Yaskawa INFORM job: R1_W70(-90,-90)KM-OK.JBI

/JOB
//NAME R1_W70(-90,-90)KM-OK
///FOLDERNAME KRIS-SCIANA
//POS
///NPOS 26,26,0,2,0,0
///TOOL 0
///POSTYPE PULSE
///PULSE
C00000=-196132,-11022,-16930,-25184,110789,12941
C00001=-198011,-10214,-12875,-25246,108327,12753
C00002=-198761,-9802,-11178,-25280,107342,12679
C00003=-197276,-7083,-6529,-24728,106458,13461
C00004=-197885,-7685,-6161,-24792,105787,13370
C00005=-197276,-7083,-6529,-24728,106458,13461
C00006=-198761,-9802,-11178,-25280,107342,12679
C00007=-193286,-14380,-9313,-33730,103593,14681
C00008=-192731,-13207,-7474,-33533,103368,14984
C00009=-193286,-14380,-9313,-33730,103593,14681
C00010=-191707,-12912,-9048,-33504,104715,14994
C00011=-204462,-13583,-17636,-16762,111010,11194
C00012=-206397,-14791,-14673,-16969,108266,10864
C00013=-206838,-12872,-13205,-17089,108253,10699
C00014=-206397,-14791,-14673,-16969,108266,10864
C00015=-200372,-41682,-38258,-22199,95841,14932
C00016=-196030,-47223,-44082,-25836,85574,-59294
C00017=-191753,-48190,-35047,-35552,77646,-65721
C00018=-174564,-4070,22503,-61552,98603,-65138
C00019=-192317,-48759,-35103,-35538,77200,-65811
C00020=-191548,-47635,-34025,-35606,77450,-65570
C00021=-178158,2617,28057,-62538,96414,-65728
C00022=-181749,10561,34999,-63443,94109,-66210
C00023=-190949,-52196,-43416,-35314,80525,-66319
C00024=-185515,-44796,-41028,-35596,84702,-65414
C00025=-121469,-118811,-94940,-10750,50157,59467
BC00000=386246,15,1075175
BC00001=386246,15,1075175
BC00002=386246,15,1075175
BC00003=386246,15,1075175
BC00004=386246,15,1075175
BC00005=386246,15,1075175
BC00006=386246,15,1075175
BC00007=386246,15,1075175
BC00008=386246,15,1075175
BC00009=386246,15,1075175
BC00010=386246,15,1075175
BC00011=386246,15,1075175
BC00012=386246,15,1075175
BC00013=386246,15,1075175
BC00014=386246,15,1075175
BC00015=386246,15,1075175
BC00016=386246,15,1075175
BC00017=385323,15,1075175
BC00018=385062,15,1075175
BC00019=385062,15,1075175
BC00020=385062,15,1075175
BC00021=385062,15,1075175
BC00022=385062,15,1075175
BC00023=377000,15,1075175
BC00024=377000,15,1075175
BC00025=219532,15,1075175
///POSTYPE BASE
///RECTAN
///RCONF 0,0,0,0,1,0,0,0,0,0,0,0,0,0,0,0,0,0,0,0,0,0,0,0
P00006=2.006,1.622,-0.565,0.0000,0.0000,0.0000
P00022=2.006,1.622,-0.565,0.0000,0.0000,0.0000
//INST
///DATE 2024/11/29 09:18
///ATTR SC,RW
///GROUP1 RB1,BS1
NOP
'r1_W70(-90,-90)
'Path S890
SFTOF
MOVJ C00000 BC00000 VJ=20.00
MOVJ C00001 BC00001 VJ=20.00
MOVL C00002 BC00002 V=100.0
MOVL C00003 BC00003 V=60.0
REFP 3 C00004 BC00004
CALL JOB:SEARCH-R1
SET P022 P006
SFTON P022
MOVL C00005 BC00005 V=60.0
MOVL C00006 BC00006 V=100.0
MOVL C00007 BC00007 V=60.0
REFP 3 C00008 BC00008
CALL JOB:SEARCH-R1
SET P022 P006
SFTON P022
MOVL C00009 BC00009 V=60.0
MOVL C00010 BC00010 V=100.0
MOVL C00011 BC00011 V=100.0
MOVL C00012 BC00012 V=60.0
REFP 3 C00013 BC00013
CALL JOB:SEARCH-R1
SET P022 P006
SFTON P022
MOVL C00014 BC00014 V=60.0
MOVL C00015 BC00015 V=100.0
MOVL C00016 BC00016 V=100.0
'Path W509
SFTOF
SFTON P022
CALL JOB:COFNIJ_DRUT
MOVJ C00017 BC00017 VJ=20.00
MOVL C00018 BC00018 V=100.0 PL=0
REFP 1 C00019 BC00019
REFP 2 C00020 BC00020
MACRO1 MJ#(0) ARGF7
ARCON
WVON WEV#(3)
MOVL C00021 BC00021 V=11.7
MOVL C00022 BC00022 V=11.7
ARCOF
WVOF
MOVL C00023 BC00023 V=166.7
MOVJ C00024 BC00024 VJ=100.00
SFTOF
MOVJ C00025 BC00025 VJ=100.00
END
